// TIA Portal V17 export
// export: Created 2025-01-08T13:55:37.1362702Z, ExportSetting WithDefaults, DisplayName Totally Integrated Automation Portal, DisplayVersion V17, DisplayName TIA Portal Openness, DisplayVersion V17, DisplayName TIA Portal Version Control Interface, DisplayVersion V17, DisplayName SINAMICS Startdrive Advanced, DisplayVersion V17 Update2, DisplayName SINAMICS Startdrive G130, G150, S120, S150, SINAMICS MV, S210, DisplayVersion V17 Update2, DisplayName SINAMICS Startdrive G110M, G120, G120C, G120D, G120P, G115D, DisplayVersion V17 Update2, DisplayName STEP 7 Professional, DisplayVersion V17, DisplayName STEP 7 Safety, DisplayVersion V17, DisplayName WinCC Advanced, DisplayVersion V17
TYPE "HSMMachineParaMask6"
// stored: IsFailsafeCompliant false
   STRUCT
      MPARA_I_Reserve_10 : Bool;
      MPARA_I_Reserve_11 : Bool;
      MPARA_I_Reserve_12 : Bool;
      MPARA_I_Reserve_13 : Bool;
      MPARA_I_Reserve_14 : Bool;
      MPARA_I_Reserve_15 : Bool;
      MPARA_I_Reserve_16 : Bool;
      MPARA_I_Reserve_17 : Bool;
      MPARA_I_Reserve_18 : Bool;
      MPARA_I_Reserve_19 : Bool;
      MPARA_I_Reserve_20 : Bool;
      MPARA_I_Reserve_21 : Bool;
      MPARA_I_Reserve_22 : Bool;
      MPARA_I_Reserve_23 : Bool;
      MPARA_I_Reserve_24 : Bool;
      MPARA_I_Reserve_25 : Bool;
   END_STRUCT;
END_TYPE
